TYPE S_General_settings :
STRUCT
	Full_speed: REAL;
	Slow_switch_speed: REAL;
END_STRUCT
END_TYPE

(* stored: Version 1.1.0.1, ProductVersion 3.1.4024.0
   DUT S_General_settings: Id {b184e8dc-311f-4adc-b3bc-f4a4e1283ebc} *)
